INTERFACE I_Arg EXTENDS __SYSTEM.IQueryInterface

END_INTERFACE

(* stored: Version 1.1.0.1
   Itf I_Arg: Id {94e755b3-19af-4e1a-a441-838a3b5f71ca} *)
